# EPICS substitutions: EX1/scr/neurons.substitutions
file network.template {
	pattern { name, name-next, in1, in2, in3, w1, w2, w3}

		{ "11", "12-sum", "01", "null", "null", "01-11", "null", "null" }
		{ "12", "13-sum", "01", "null", "null", "01-12", "null", "null" }
		{ "13", "21-sum", "01", "null", "null", "01-13", "null", "null"  }

		{ "21", "22-sum", "11", "12", "13", "11-21", "12-21", "13-21" }
		{ "22", "23-sum", "11", "12", "13", "11-22", "12-22", "13-22" }
		{ "23", "score-fanout", "11", "12", "13", "11-23", "12-23", "13-23" }
}

file softmax.template {
	pattern { name, other1, other2 }
		{ "21", "22", "23" }
		{ "22", "21", "23" }
		{ "23", "21", "22" }
}

file weights.template {
	pattern { name1, name2, weight }
		{ "01", "11", "-20" }
		{ "01", "12", "20" }
		{ "01", "13", "20" }

		{ "11", "21", "6" }
		{ "12", "21", "0" }
		{ "13", "21", "0" }

		{ "11", "22", "0" }
		{ "12", "22", "6" }
		{ "13", "22", "-6" }

		{ "11", "23", "0" }
		{ "12", "23", "0" }
		{ "13", "23", "6" }
}

file bias.template {
	pattern { name, bias }

		{ "11", "6.6" }
		{ "12", "-6.6" }
		{ "13", "-13.2" }

		{ "21", "-3" }
		{ "22", "-3" }
		{ "23", "-3" }
}
